{attribute addProperty BoxType "KL9110"}
{attribute addProperty Id "PowerAT %I*BOOL000ShortCircuitAT %I*BOOL000"}
{attribute addProperty CRC "158341521"}
{attribute addProperty SizeInBites "0"}
{attribute addProperty SizeInBytes "0"}
TYPE Channel_09701991 :
STRUCT
	{attribute addProperty Name "Power"}
	Power AT %I* : BOOL;
	{attribute addProperty Name "ShortCircuit"}
	ShortCircuit AT %I* : BOOL;
END_STRUCT
END_TYPE

(* stored: Version 1.2.0.0, ProductVersion 3.1.4024.9
   DUT Channel_09701991: Id {af5ebe83-fcf4-45e7-93a4-e1bd1c6f7a96} *)
